Staubli VAL3: CloseSingnal.pgx

program CloseSingnal()
begin
  //
  IO:dOut["dOut4"]=false
end
